TYPE ST_HMI_TempController_Config :
STRUCT
	Param: ST_Param_TempController;
END_STRUCT
END_TYPE

(* stored: Version 1.1.0.1, ProductVersion 3.1.4024.12
   DUT ST_HMI_TempController_Config: Id {9cc125f6-1992-49ee-a973-8c4ecf1e5b63} *)
